// ---- 03_ControlPrimitives/Stamp/Stamp_StampWorkpiece.TcPOU
FUNCTION_BLOCK Stamp_StampWorkpiece EXTENDS ControlPrimitiveBase
VAR_INPUT
END_VAR
VAR_OUTPUT
END_VAR
VAR
	// (EProcessVariables.Stamp_WorkpieceState = 1) AND (EProcessVariables.Stamp_WPAtStamp = TRUE)
// 	m_compExpr273: ComparisonExpression(EProcessVariables.Stamp_WorkpieceState, EComparisonType.equals, EDataType.numeric, FALSE, 1, '', TRUE);
	m_precondition: ComparisonExpression(EProcessVariables.Stamp_WPAtStamp, EComparisonType.equals, EDataType.binary, TRUE, 0, '', TRUE);
// 	m_precondition: BoolExpression(m_compExpr273, EBoolOperation.and_op, m_compExpr275);
	
	// EProcessVariables.Stamp_WorkpieceState = 2
	m_postcondition: ComparisonExpression(EProcessVariables.Stamp_WorkpieceState, EComparisonType.equals, EDataType.numeric, FALSE, 2, '', TRUE);

	m_ptrStamp: POINTER TO Stamp;
	
	m_step: INT := 0;
	t_Stamp : TON;
END_VAR

SUPER^();

METHOD Abort : BOOL
VAR_INPUT
END_VAR
m_ptrStamp^.m_stampingCylinder.METH_Retract();
m_ptrStamp^.m_slidingCylinder.METH_Extend();
Abort := TRUE;
END_METHOD

(* Execution logic of this Control Primitive. *)
METHOD PROTECTED ExecuteInternal : BOOL
VAR_INPUT
	(*
	 * pressure_white: INT
	 * pressure_black: INT
	 * pressure_metal: INT
	 *)
	i_params: ParameterSet;
END_VAR
VAR
	m_pressureVal: SValue;
END_VAR
ExecuteInternal := FALSE;

CASE m_step OF
	0: // take in wp
	m_ptrStamp^.m_slidingCylinder.METH_Retract();
	IF m_ptrStamp^.m_slidingCylinder.Retracted THEN
		m_step := 1;
	END_IF
	
	1: // stamp wp
	m_ptrStamp^.StampPressure := GetPressure(i_params);
	m_ptrStamp^.m_stampingCylinder.METH_Extend();
	t_Stamp(IN:=TRUE, PT:=T#1500MS);
	IF t_Stamp.Q THEN
		IF m_ptrStamp^.StampPressure >= m_pressureVal.Value.Numeric THEN
			m_step := 2;
			t_Stamp(IN:=FALSE);
		END_IF
	END_IF
	
	2: // retract stamp
	m_ptrStamp^.m_stampingCylinder.METH_Retract();
	IF m_ptrStamp^.m_stampingCylinder.Retracted THEN
		m_step := 3;
	END_IF
	
	3: // provide wp
	m_ptrStamp^.m_slidingCylinder.METH_Extend();
	IF m_ptrStamp^.m_slidingCylinder.Extended THEN
		m_step := 0;
		ExecuteInternal := TRUE;
	END_IF
END_CASE
END_METHOD

METHOD FB_init : BOOL
VAR_INPUT
	bInitRetains : BOOL; // if TRUE, the retain variables are initialized (warm start / cold start)
	bInCopyCode : BOOL;  // if TRUE, the instance afterwards gets moved into the copy code (online change)
	
	i_ptrStamp: POINTER TO Stamp;
END_VAR
m_ptrStamp := i_ptrStamp;

m_id := EPrimitives.Stamp_StampWorkpiece;
m_timeout := T#200S;
m_paramDefinition := 'pressure_white:INT;pressure_black:INT;pressure_metal:INT;';

Precondition := m_precondition;
Postcondition := m_postcondition;
END_METHOD

METHOD PRIVATE GetPressure : INT
VAR_INPUT
	(*
	 * pressure_white: INT
	 * pressure_black: INT
	 * pressure_metal: INT
	 *)
	i_params: ParameterSet;
END_VAR
VAR
	m_pressureVal: SValue;
END_VAR
CASE LREAL_TO_UINT(m_st^.GetNumeric(EProcessVariables.Stamp_ProductType)) OF
	EProductTypes.white:
		m_pressureVal := i_params.Retrieve('pressure_white');
		GetPressure := LREAL_TO_INT(m_pressureVal.Value.Numeric);
	EProductTypes.black:
		m_pressureVal := i_params.Retrieve('pressure_black');
		GetPressure := LREAL_TO_INT(m_pressureVal.Value.Numeric);
	EProductTypes.metal:
		m_pressureVal := i_params.Retrieve('pressure_metal');
		GetPressure := LREAL_TO_INT(m_pressureVal.Value.Numeric);
	ELSE
		GetPressure := 0;
END_CASE
END_METHOD

END_FUNCTION_BLOCK

// ---- 05_HardwareControl/EquipmentModule/Stamps/Stamp.TcPOU
FUNCTION_BLOCK Stamp EXTENDS BaseComponent
VAR_INPUT
END_VAR
VAR_OUTPUT
END_VAR
VAR
	m_stampingCylinder: MonostableCylinder;
	m_slidingCylinder: BistableCylinder;
	m_pressureValve: PropotionalValve;
	
	m_presenceSensor: PresenceSensor;
	m_pressureSensor: PressureSensor;
END_VAR

PROPERTY StampPressure : INT
GET
StampPressure:=m_pressureSensor.Value;
END_GET
SET
m_pressureValve.Pressure := StampPressure;
END_SET
END_PROPERTY

PROPERTY WPAtStart : BOOL
GET
WPAtStart := m_presenceSensor.Value;
END_GET
END_PROPERTY

END_FUNCTION_BLOCK

// ---- 05_HardwareControl/ControlModule/Pushers/BistableCylinder.TcPOU
FUNCTION_BLOCK BistableCylinder EXTENDS BaseCylinder
VAR_INPUT	
END_VAR
VAR_OUTPUT
END_VAR
VAR	
	//Hardware
	DO_Retract AT %Q* : BOOL;
END_VAR

METHOD METH_Extend : BOOL
DO_Extend := TRUE;
DO_Retract := FALSE;
END_METHOD

METHOD METH_Retract : BOOL
DO_Extend := FALSE;
DO_Retract := TRUE;
END_METHOD

END_FUNCTION_BLOCK

// ---- 05_HardwareControl/ControlModule/Valves/PropotionalValve.TcPOU
FUNCTION_BLOCK PropotionalValve
VAR_INPUT
END_VAR
VAR_OUTPUT
END_VAR
VAR
	//Hardware
	AO_SetPressure AT %Q* : INT;
END_VAR

PROPERTY Pressure : INT
SET
AO_SetPressure := Pressure;
END_SET
END_PROPERTY

END_FUNCTION_BLOCK

// ---- 05_HardwareControl/ControlModule/Sensors/PressureSensor.TcPOU
FUNCTION_BLOCK PressureSensor IMPLEMENTS ITF_AnalogSensor
VAR_INPUT
END_VAR
VAR_OUTPUT
END_VAR
VAR
	//Hardware
	AI_CurrentPressure AT %I* : INT;
END_VAR

PROPERTY Value : INT
GET
Value := AI_CurrentPressure;
END_GET
END_PROPERTY

END_FUNCTION_BLOCK

// ---- 04_HardwareObservation/ObserveCrane.TcPOU
FUNCTION_BLOCK ObserveCrane EXTENDS HardwareObservationBase
VAR_INPUT
END_VAR
VAR_OUTPUT
END_VAR
VAR
	m_ptrCrane: POINTER TO Crane;
	m_ptrCraneWP: POINTER TO xPPUProduct;
	
	m_rtAtStack: R_TRIG;
	m_rtAtLSC: R_TRIG;
	m_rtAtStamp: R_TRIG;
	
	m_resetCranePos: BOOL;
	
	// needed for a regression for the analog AngleDeg
	poti0: REAL;
	poti90: REAL;
	poti180: REAL;
END_VAR

METHOD FB_init : BOOL
VAR_INPUT
	bInitRetains : BOOL; // if TRUE, the retain variables are initialized (warm start / cold start)
	bInCopyCode : BOOL;  // if TRUE, the instance afterwards gets moved into the copy code (online change)

	i_ptrCrane: POINTER TO Crane;
	i_ptrWP: POINTER TO xPPUProduct;
END_VAR
m_ptrCrane := i_ptrCrane;
m_ptrCraneWP := i_ptrWP;
END_METHOD

METHOD  ResetDefinition : BOOL
VAR_INPUT
END_VAR
m_resetCranePos := TRUE;
END_METHOD

(* Update an instance of ProcessState with the part of the process that can be observed by this Hardware Interface. *)
METHOD UpdateProcessObservation : BOOL
VAR_IN_OUT
	io_processState: ProcessState;
END_VAR
VAR
	potiVal: REAL;
	x_bar: REAL;
	y_bar: REAL;
	a: REAL := -88.16748;		// initial value (calibrated 30 April 2025)
	b: REAL := 0.0129453959;	// initial value (calibrated 30 April 2025)
END_VAR
io_processState.UpdateState_Binary(EProcessVariables.Crane_AtStack, m_ptrCrane^.AtStack, i_force := TRUE);
io_processState.UpdateState_Binary(EProcessVariables.Crane_AtStamp, m_ptrCrane^.AtStamp, i_force := TRUE);
io_processState.UpdateState_Binary(EProcessVariables.Crane_AtLSC, m_ptrCrane^.AtConveyor, i_force := TRUE);
io_processState.UpdateState_Binary(EProcessVariables.Crane_HoldingWorkpiece, m_ptrCrane^.o_VacuumGripper.WPTaken, i_force := TRUE);
io_processState.UpdateState_Binary(EProcessVariables.Crane_CylinderExtended, m_ptrCrane^.o_MonostableCylinder.Extended, i_force := TRUE);
io_processState.UpdateState_Binary(EProcessVariables.Crane_CylinderRetracted, m_ptrCrane^.o_MonostableCylinder.Retracted, i_force := TRUE);

// Angle [in degrees] regression
potiVal := m_ptrCrane^.Motor.AI_Position;
IF m_ptrCrane^.AtStack THEN
	poti0 := potiVal;
ELSIF m_ptrCrane^.AtConveyor THEN
	poti90 := potiVal;
ELSIF m_ptrCrane^.AtStamp THEN
	poti180 := potiVal;
END_IF

IF poti0 <> 0 AND poti90 <> 0 AND poti180 <> 0 THEN
	x_bar := (poti0 + poti90 + poti180) / 3;
	y_bar := (90+180)/3;
	b := ((poti0 - x_bar)*-y_bar + (poti90 - x_bar)*(90 - y_bar) + (poti180 - x_bar)*(180 - y_bar))/
		(EXPT(poti0 - x_bar, 2) + EXPT(poti90 - x_bar, 2) + EXPT(poti180 - x_bar, 2));
	a := y_bar - b*x_bar;
ELSIF poti0 <> 0 AND poti90 <> 0 THEN
	x_bar := (poti0 + poti90) / 2;
	y_bar := 90/2;
	b := ((poti0 - x_bar)*-y_bar + (poti90 - x_bar)*(90 - y_bar))/
		(EXPT(poti0 - x_bar, 2) + EXPT(poti90 - x_bar, 2));
	a := y_bar - b*x_bar;
ELSIF poti90 <> 0 AND poti180 <> 0 THEN
	x_bar := (poti90 + poti180) / 2;
	y_bar := (90+180)/2;
	b := ((poti90 - x_bar)*(90 - y_bar) + (poti180 - x_bar)*(180 - y_bar))/
		(EXPT(poti90 - x_bar, 2) + EXPT(poti180 - x_bar, 2));
	a := y_bar - b*x_bar;
END_IF

io_processState.UpdateState_Numeric(EProcessVariables.Crane_Angle, a + b*potiVal, i_force := TRUE);

m_rtAtStack(CLK := m_ptrCrane^.AtStack);
m_rtAtStamp(CLK := m_ptrCrane^.AtStamp);
m_rtAtLSC(CLK := m_ptrCrane^.AtConveyor);

IF m_rtAtStack.Q OR m_rtAtStamp.Q OR m_rtAtLSC.Q THEN
	io_processState.UpdateState_Defined(EProcessVariables.Crane_AtStack, TRUE);
	io_processState.UpdateState_Defined(EProcessVariables.Crane_AtStamp, TRUE);
	io_processState.UpdateState_Defined(EProcessVariables.Crane_AtLSC, TRUE);
END_IF
IF m_resetCranePos THEN
	io_processState.UpdateState_Defined(EProcessVariables.Crane_AtStack, FALSE);
	io_processState.UpdateState_Defined(EProcessVariables.Crane_AtStamp, FALSE);
	io_processState.UpdateState_Defined(EProcessVariables.Crane_AtLSC, FALSE);
	m_resetCranePos := FALSE;
END_IF

io_processState.UpdateState_Defined(EProcessVariables.Crane_HoldingWorkpiece, TRUE);
io_processState.UpdateState_Defined(EProcessVariables.Crane_CylinderExtended, TRUE);
io_processState.UpdateState_Defined(EProcessVariables.Crane_CylinderRetracted, TRUE);
io_processState.UpdateState_Defined(EProcessVariables.Crane_Angle, TRUE);
END_METHOD

END_FUNCTION_BLOCK

// ---- 04_HardwareObservation/xPPUProduct.TcPOU
FUNCTION_BLOCK xPPUProduct EXTENDS ProductBase
VAR CONSTANT
	LIGHT_IDX: USINT := 1;
	METAL_IDX: USINT := 2;
	PRESENT_IDX: USINT := 3;
	STAMPED_IDX: USINT := 4;

	LIGHT_MASK: BYTE := 2#0000_0001;
	METAL_MASK: BYTE := 2#0000_0010;
	PRESENT_MASK: BYTE := 2#0000_0100;
	STAMPED_MASK: BYTE := 2#0000_1000;
END_VAR
VAR
	m_productStampedIdx: UINT;
END_VAR

//FB_Init is always available implicitly and it is used primarily for initialization.
//The return value is not evaluated. For a specific influence, you can also declare the
//methods explicitly and provide additional code there with the standard initialization
//code. You can evaluate the return value.
METHOD FB_Init: BOOL
VAR_INPUT
    bInitRetains: BOOL; // TRUE: the retain variables are initialized (reset warm / reset cold)
    bInCopyCode: BOOL;  // TRUE: the instance will be copied to the copy code afterward (online change)
	
	i_productTypeVarId: UINT;
	i_productStampedVarId: UINT;
END_VAR
// set the variable indices (on remote, the RA does this)
raIn_processStateIdx := i_productTypeVarId;

m_productStampedIdx := i_productStampedVarId;

// set the variables' data types
m_vals[RES_IDX].DataType := EDataType.numeric;
m_vals[LIGHT_IDX].DataType := EDataType.binary;
m_vals[METAL_IDX].DataType := EDataType.binary;
m_vals[PRESENT_IDX].DataType := EDataType.binary;
END_METHOD

PROPERTY IsLight : BOOL
GET
IsLight := m_vals[LIGHT_IDX].Defined AND m_vals[LIGHT_IDX].Value.Binary;
END_GET
SET
m_vals[LIGHT_IDX].DataType := EDataType.binary;
m_vals[LIGHT_IDX].Defined := TRUE;
m_vals[LIGHT_IDX].Value.Binary := IsLight;

UpdateMaterial();
END_SET
END_PROPERTY

PROPERTY IsMetal : BOOL
GET
IsMetal := m_vals[METAL_IDX].Defined AND m_vals[METAL_IDX].Value.Binary;
END_GET
SET
m_vals[METAL_IDX].DataType := EDataType.binary;
m_vals[METAL_IDX].Defined := TRUE;
m_vals[METAL_IDX].Value.Binary := IsMetal;

UpdateMaterial();
END_SET
END_PROPERTY

PROPERTY IsPresent : BOOL
GET
IsPresent := m_vals[PRESENT_IDX].Defined AND m_vals[PRESENT_IDX].Value.Binary;
END_GET
SET
m_vals[PRESENT_IDX].DataType := EDataType.binary;
m_vals[PRESENT_IDX].Defined := TRUE;
m_vals[PRESENT_IDX].Value.Binary := IsPresent;

UpdateMaterial();
END_SET
END_PROPERTY

PROPERTY IsStamped : BOOL
GET
IsStamped := m_vals[STAMPED_IDX].Defined AND m_vals[STAMPED_IDX].Value.Binary;
END_GET
SET
m_vals[STAMPED_IDX].DataType := EDataType.binary;
m_vals[STAMPED_IDX].Defined := TRUE;
m_vals[STAMPED_IDX].Value.Binary := IsStamped;

UpdateMaterial();
END_SET
END_PROPERTY

(* Based on the aggregated product type value, set the separete input values for a consistent shift register. *)
METHOD ReverseSetInputs : BOOL
VAR
	res: BYTE;
END_VAR
res := LREAL_TO_BYTE(m_vals[RES_IDX].Value.Numeric);

m_vals[LIGHT_IDX].Value.Binary := (res AND LIGHT_MASK) <> 0;
m_vals[METAL_IDX].Value.Binary := (res AND METAL_MASK) <> 0;
m_vals[PRESENT_IDX].Value.Binary := (res AND PRESENT_MASK) <> 0;
m_vals[STAMPED_IDX].Value.Binary := (res AND STAMPED_MASK) <> 0;

m_vals[LIGHT_IDX].Defined := TRUE;
m_vals[METAL_IDX].Defined := TRUE;
m_vals[PRESENT_IDX].Defined := TRUE;
m_vals[STAMPED_IDX].Defined := TRUE;
END_METHOD

METHOD PRIVATE UpdateMaterial : BOOL
VAR
	res: BYTE;
END_VAR
// use separate bits to encode the product info
res := 2#0000_0000;

IF IsLight THEN
	res := res OR LIGHT_MASK;
END_IF
IF IsMetal THEN
	res := res OR METAL_MASK;
END_IF
IF IsPresent THEN
	res := res OR PRESENT_MASK;
END_IF
IF IsStamped THEN
	res := res OR STAMPED_MASK;
END_IF

m_vals[RES_IDX].DataType := EDataType.numeric;
m_vals[RES_IDX].Defined := TRUE;
m_vals[RES_IDX].Value.Numeric := BYTE_TO_LREAL(res);
END_METHOD

METHOD PROTECTED UpdateProcessObsInternal : BOOL
VAR_IN_OUT
	io_processState: ProcessState;
END_VAR
VAR
	prodType: EProductTypes;
END_VAR
IF NOT IsLight AND NOT IsMetal AND NOT IsPresent THEN
	prodType := EProductTypes.none;
ELSIF IsLight AND NOT IsMetal AND IsPresent THEN
	prodType := EProductTypes.white;
ELSIF NOT IsLight AND NOT IsMetal AND IsPresent THEN
	prodType := EProductTypes.black;
ELSIF IsMetal AND IsPresent THEN
	prodType := EProductTypes.metal;
END_IF

io_processState.UpdateState_Numeric(raIn_processStateIdx, UINT_TO_LREAL(prodType), i_force := TRUE);
io_processState.UpdateState_Binary(m_productStampedIdx, IsStamped, i_force := TRUE);

io_processState.UpdateState_Defined(raIn_processStateIdx, TRUE);
io_processState.UpdateState_Defined(m_productStampedIdx, TRUE);
END_METHOD

END_FUNCTION_BLOCK

// ---- 04_HardwareObservation/ObserveLSC.TcPOU
FUNCTION_BLOCK ObserveLSC EXTENDS HardwareObservationBase
VAR_INPUT
END_VAR
VAR_OUTPUT
END_VAR
VAR
	m_ptrLSC: POINTER TO LargeSortingConveyor;
	m_ptrLSCWP: POINTER TO xPPUProduct;
	
	m_rtAtStart: R_TRIG;
	m_rtLightAtStart: R_TRIG;
	m_rtLightAtMid: R_TRIG;
	m_rtLightAtEnd: R_TRIG;
	m_rtMetalAtStart: R_TRIG;
	m_rtMetalAtMid: R_TRIG;
	m_rtWpAtRampStart: R_TRIG;
	m_rtWpAtRampMiddle: R_TRIG;
	m_rtWpAtRampEnd: R_TRIG;
	
	m_LSCemptytimeout: TON;
	m_resetProductDefined: BOOL;
	
	m_didInit: BOOL := FALSE;
END_VAR

METHOD FB_init : BOOL
VAR_INPUT
	bInitRetains : BOOL; // if TRUE, the retain variables are initialized (warm start / cold start)
	bInCopyCode : BOOL;  // if TRUE, the instance afterwards gets moved into the copy code (online change)

	i_ptrLSC: POINTER TO LargeSortingConveyor;
	i_ptrWP: POINTER TO xPPUProduct;
END_VAR
m_ptrLSC := i_ptrLSC;
m_ptrLSCWP := i_ptrWP;
END_METHOD

METHOD  ResetDefinition : BOOL
VAR_INPUT
END_VAR
m_resetProductDefined := TRUE;
END_METHOD

(* Update an instance of ProcessState with the part of the process that can be observed by this Hardware Interface. *)
METHOD UpdateProcessObservation : BOOL
VAR_IN_OUT
	io_processState: ProcessState;
END_VAR
m_rtAtStart(CLK := m_ptrLSC^.WPAtStart);
m_rtLightAtStart(CLK := m_ptrLSC^.LightWPAtStart);
m_rtLightAtMid(CLK := m_ptrLSC^.LightWPAtMid);
m_rtLightAtEnd(CLK := m_ptrLSC^.LightWPAtEnd);
m_rtMetalAtStart(CLK := m_ptrLSC^.MetalWPAtStart);
m_rtMetalAtMid(CLK := m_ptrLSC^.MetalWPAtMid);
m_rtWpAtRampStart(CLK := m_ptrLSC^.WPAtRampStart);
m_rtWpAtRampMiddle(CLK := m_ptrLSC^.WPAtRampMiddle);
m_rtWpAtRampEnd(CLK := m_ptrLSC^.WPAtRampEnd);

io_processState.UpdateState_Binary(EProcessVariables.LSC_WorkpieceAtEntry, m_ptrLSC^.WPAtStart, TRUE);
io_processState.UpdateState_Binary(EProcessVariables.LSC_WPAtRampStart, m_ptrLSC^.WPAtRampStart, TRUE);
io_processState.UpdateState_Binary(EProcessVariables.LSC_WPAtRampMiddle, m_ptrLSC^.WPAtRampMiddle, TRUE);
io_processState.UpdateState_Binary(EProcessVariables.LSC_WPAtRampEnd, m_ptrLSC^.WPAtRampEnd, TRUE);
io_processState.UpdateState_Binary(EProcessVariables.LSC_SwitchExtended, m_ptrLSC^.m_Switch.Extended, TRUE);
io_processState.UpdateState_Binary(EProcessVariables.LSC_SwitchRetracted, m_ptrLSC^.m_Switch.Retracted, TRUE);
io_processState.UpdateState_Binary(EProcessVariables.LSC_WPAtInductiveSensorEnd, m_ptrLSC^.MetalWPAtMid, TRUE);

IF NOT m_didInit THEN
	io_processState.UpdateState_Numeric(EProcessVariables.LSC_RampStartWPCount, 0, TRUE);
	io_processState.UpdateState_Numeric(EProcessVariables.LSC_RampMiddleWPCount, 0, TRUE);
	io_processState.UpdateState_Numeric(EProcessVariables.LSC_RampEndWPCount, 0, TRUE);
	m_didInit := TRUE;
END_IF

IF m_rtWpAtRampStart.Q THEN
	io_processState.UpdateState_NumericIncrement(EProcessVariables.LSC_RampStartWPCount, TRUE);
END_IF
IF m_rtWpAtRampMiddle.Q THEN
	io_processState.UpdateState_NumericIncrement(EProcessVariables.LSC_RampMiddleWPCount, TRUE);
END_IF
IF m_rtWpAtRampEnd.Q THEN
	io_processState.UpdateState_NumericIncrement(EProcessVariables.LSC_RampEndWPCount, TRUE);
END_IF

io_processState.UpdateState_Defined(EProcessVariables.LSC_WorkpieceAtEntry, TRUE);
io_processState.UpdateState_Defined(EProcessVariables.LSC_WPAtRampStart, TRUE);
io_processState.UpdateState_Defined(EProcessVariables.LSC_WPAtRampMiddle, TRUE);
io_processState.UpdateState_Defined(EProcessVariables.LSC_WPAtRampEnd, TRUE);
io_processState.UpdateState_Defined(EProcessVariables.LSC_SwitchExtended, TRUE);
io_processState.UpdateState_Defined(EProcessVariables.LSC_SwitchRetracted, TRUE);
io_processState.UpdateState_Defined(EProcessVariables.LSC_WPAtInductiveSensorEnd, TRUE);
// TODO - the following are technically not defined but how can we avoid that?
io_processState.UpdateState_Defined(EProcessVariables.LSC_RampStartWPCount, TRUE);
io_processState.UpdateState_Defined(EProcessVariables.LSC_RampMiddleWPCount, TRUE);
io_processState.UpdateState_Defined(EProcessVariables.LSC_RampEndWPCount, TRUE);

// update WP info (if there are sensors available), then update the process variables list
IF m_rtAtStart.Q THEN
	m_ptrLSCWP^.IsPresent := TRUE;
END_IF
IF m_rtLightAtStart.Q OR m_rtLightAtMid.Q OR m_rtLightAtEnd.Q THEN
	m_ptrLSCWP^.IsLight := TRUE;
END_IF
IF m_rtMetalAtStart.Q OR m_rtMetalAtMid.Q THEN
	m_ptrLSCWP^.IsMetal := TRUE;
END_IF

// reset IsPresent if any of the ramps are triggered
IF m_ptrLSC^.WPAtRampStart OR m_ptrLSC^.WPAtRampMiddle OR m_ptrLSC^.WPAtRampEnd THEN
	m_ptrLSCWP^.IsPresent := FALSE;
END_IF

//if the conveyor moves forward for a certain time, it has to empty, therefore LSCProductType is defined
IF m_ptrLSC^.Motor.TurningClockwise THEN
	m_LSCemptytimeout(IN:= TRUE, PT:=T#3500MS);
ELSE
	m_LSCemptytimeout(IN:= FALSE);
END_IF

IF m_LSCemptytimeout.Q THEN
	io_processState.UpdateState_Defined(EProcessVariables.LSC_ProductType, TRUE);
	m_LSCemptytimeout(IN:= FALSE);
END_IF

IF m_resetProductDefined THEN
	m_resetProductDefined := TRUE;
END_IF
END_METHOD

END_FUNCTION_BLOCK

// ---- 04_HardwareObservation/ObservePAC.TcPOU
FUNCTION_BLOCK ObservePAC EXTENDS HardwareObservationBase
VAR_INPUT
END_VAR
VAR_OUTPUT
END_VAR
VAR
	m_ptrPAC: POINTER TO PicAlphaConveyor;
	m_ptrPACWP1: POINTER TO xPPUProduct;
	m_ptrPACWP2: POINTER TO xPPUProduct;
	m_ptrPACWP3: POINTER TO xPPUProduct;
END_VAR

METHOD FB_init : BOOL
VAR_INPUT
	bInitRetains : BOOL; // if TRUE, the retain variables are initialized (warm start / cold start)
	bInCopyCode : BOOL;  // if TRUE, the instance afterwards gets moved into the copy code (online change)
	
	i_ptrPAC: POINTER TO PicAlphaConveyor;
	i_ptrWP1: POINTER TO xPPUProduct;
	i_ptrWP2: POINTER TO xPPUProduct;
	i_ptrWP3: POINTER TO xPPUProduct;

	
END_VAR
m_ptrPAC := i_ptrPAC;
m_ptrPACWP1 := i_ptrWP1;
m_ptrPACWP2 := i_ptrWP2;
m_ptrPACWP3 := i_ptrWP3;
END_METHOD

METHOD  ResetDefinition : BOOL
VAR_INPUT
END_VAR
;
END_METHOD

(* Update an instance of ProcessState with the part of the process that can be observed by this Hardware Interface. *)
METHOD UpdateProcessObservation : BOOL
VAR_IN_OUT
	io_processState: ProcessState;
END_VAR
io_processState.UpdateState_Binary(EProcessVariables.PAC_WPAtStart, m_ptrPAC^.WPAtStart, TRUE);
io_processState.UpdateState_Binary(EProcessVariables.PAC_WPAtEnd, m_ptrPAC^.WPAtEnd, TRUE);
io_processState.UpdateState_Binary(EProcessVariables.PAC_SwitchExtended, m_ptrPAC^.m_Switch.Extended, TRUE);
io_processState.UpdateState_Binary(EProcessVariables.PAC_SwitchRetracted, m_ptrPAC^.m_Switch.Retracted, TRUE);
io_processState.UpdateState_Numeric(EProcessVariables.PAC_WPNumber, INT_TO_LREAL(m_ptrPAC^.m_WPNumberAtPAC), TRUE);

io_processState.UpdateState_Defined(EProcessVariables.PAC_WPAtStart, TRUE);
io_processState.UpdateState_Defined(EProcessVariables.PAC_WPAtEnd, TRUE);
io_processState.UpdateState_Defined(EProcessVariables.PAC_SwitchExtended, TRUE);
io_processState.UpdateState_Defined(EProcessVariables.PAC_SwitchRetracted, TRUE);
io_processState.UpdateState_Defined(EProcessVariables.PAC_WPNumber, TRUE);
END_METHOD

END_FUNCTION_BLOCK

// ---- 04_HardwareObservation/ObservePicAlpha.TcPOU
FUNCTION_BLOCK ObservePicAlpha EXTENDS HardwareObservationBase
VAR_INPUT
END_VAR
VAR_OUTPUT
END_VAR
VAR
	m_ptrPicAlpha: POINTER TO PicAlpha;
	m_ptrPicAlphaWP: POINTER TO xPPUProduct;

	m_PicAlphaPosDefinedState: BOOL := FALSE;
END_VAR

METHOD FB_init : BOOL
VAR_INPUT
	bInitRetains : BOOL; // if TRUE, the retain variables are initialized (warm start / cold start)
	bInCopyCode : BOOL;  // if TRUE, the instance afterwards gets moved into the copy code (online change)
	
	i_ptrPicAlpha: POINTER TO PicAlpha;
	i_ptrWP: POINTER TO xPPUProduct;
END_VAR
m_ptrPicAlpha := i_ptrPicAlpha;
m_ptrPicAlphaWP := i_ptrWP;
END_METHOD

METHOD  ResetDefinition : BOOL
VAR_INPUT
END_VAR
m_PicAlphaPosDefinedState := FALSE;
END_METHOD

(* Update an instance of ProcessState with the part of the process that can be observed by this Hardware Interface. *)
METHOD UpdateProcessObservation : BOOL
VAR_IN_OUT
	io_processState: ProcessState;
END_VAR
VAR
	m_sensorCount : UINT;
END_VAR
io_processState.UpdateState_Binary(EProcessVariables.PicAlpha_AtPos1, m_ptrPicAlpha^.PresenceSensorPosition1Value, i_force := TRUE);
io_processState.UpdateState_Binary(EProcessVariables.PicAlpha_AtPos2, m_ptrPicAlpha^.PresenceSensorPosition2Value, i_force := TRUE);
io_processState.UpdateState_Binary(EProcessVariables.PicAlpha_AtPos3, m_ptrPicAlpha^.PresenceSensorPosition3Value, i_force := TRUE);
io_processState.UpdateState_Binary(EProcessVariables.PicAlpha_AtPos4, m_ptrPicAlpha^.PresenceSensorPosition4Value, i_force := TRUE);
io_processState.UpdateState_Binary(EProcessVariables.PicAlpha_HoldingWorkpiece, m_ptrPicAlpha^.o_VacuumGripper.WPTaken, i_force := TRUE);
io_processState.UpdateState_Binary(EProcessVariables.PicAlpha_CylinderExtended, m_ptrPicAlpha^.o_MonostableCylinder.Extended, i_force := TRUE);
io_processState.UpdateState_Binary(EProcessVariables.PicAlpha_CylinderRetracted, m_ptrPicAlpha^.o_MonostableCylinder.Retracted, i_force := TRUE);
io_processState.UpdateState_Numeric(EProcessVariables.PicAlpha_Distance, INT_TO_LREAL(m_ptrPicAlpha^.o_Distance), i_force := TRUE);

io_processState.UpdateState_Defined(EProcessVariables.PicAlpha_HoldingWorkpiece, TRUE);
io_processState.UpdateState_Defined(EProcessVariables.PicAlpha_CylinderExtended, TRUE);
io_processState.UpdateState_Defined(EProcessVariables.PicAlpha_CylinderRetracted, TRUE);
io_processState.UpdateState_Defined(EProcessVariables.PicAlpha_Distance, TRUE);

// update WP info (if there are sensors available), then update the process variables list

IF m_ptrPicAlpha^.PresenceSensorPosition3Value AND NOT (m_ptrPicAlpha^.PresenceSensorPosition1Value OR m_ptrPicAlpha^.PresenceSensorPosition2Value OR m_ptrPicAlpha^.PresenceSensorPosition4Value) THEN
	m_PicAlphaPosDefinedState :=  TRUE;
END_IF
IF m_PicAlphaPosDefinedState THEN
	m_sensorCount := 0;	
END_IF
IF m_ptrPicAlpha^.PresenceSensorPosition1Value OR m_ptrPicAlpha^.PresenceSensorPosition2Value THEN
 	m_sensorCount := m_sensorCount + 1;
END_IF
IF m_ptrPicAlpha^.PresenceSensorPosition3Value THEN
 	m_sensorCount := m_sensorCount + 1;
END_IF
IF m_ptrPicAlpha^.PresenceSensorPosition4Value THEN
 	m_sensorCount := m_sensorCount + 1;
END_IF

IF m_sensorCount > 1 THEN // if more than one sensor is pressed at the same time, the position is undefined
	m_PicAlphaPosDefinedState := FALSE;	
END_IF

io_processState.UpdateState_Defined(EProcessVariables.PicAlpha_AtPos1, m_PicAlphaPosDefinedState);
io_processState.UpdateState_Defined(EProcessVariables.PicAlpha_AtPos2, m_PicAlphaPosDefinedState);
io_processState.UpdateState_Defined(EProcessVariables.PicAlpha_AtPos3, m_PicAlphaPosDefinedState);
io_processState.UpdateState_Defined(EProcessVariables.PicAlpha_AtPos4, m_PicAlphaPosDefinedState);
END_METHOD

END_FUNCTION_BLOCK

// ---- 04_HardwareObservation/ObserveRFC.TcPOU
FUNCTION_BLOCK ObserveRFC
VAR_INPUT
END_VAR
VAR_OUTPUT
END_VAR
VAR
	m_ptrRFC: POINTER TO RefeedingConveyor;
	m_ptrRFCWP1: POINTER TO xPPUProduct;
	m_ptrRFCWP2: POINTER TO xPPUProduct;
END_VAR

METHOD FB_init : BOOL
VAR_INPUT
	bInitRetains : BOOL; // if TRUE, the retain variables are initialized (warm start / cold start)
	bInCopyCode : BOOL;  // if TRUE, the instance afterwards gets moved into the copy code (online change)
	
	i_ptrRFC: POINTER TO RefeedingConveyor;
	i_ptrWP1: POINTER TO xPPUProduct;
	i_ptrWP2: POINTER TO xPPUProduct;
END_VAR
m_ptrRFC := i_ptrRFC;
m_ptrRFCWP1 := i_ptrWP1;
m_ptrRFCWP2 := i_ptrWP2;
END_METHOD

METHOD ResetDefinition : BOOL
VAR_INPUT
END_VAR
;
END_METHOD

(* Update an instance of ProcessState with the part of the process that can be observed by this Hardware Interface. *)
METHOD UpdateProcessObservation : BOOL
VAR_IN_OUT
	io_processState: ProcessState;
END_VAR
io_processState.UpdateState_Binary(EProcessVariables.RFC_WPAtStart, m_ptrRFC^.WPAtStart, TRUE);
io_processState.UpdateState_Binary(EProcessVariables.RFC_WPAtEnd, m_ptrRFC^.WPAtEnd, TRUE);
io_processState.UpdateState_Binary(EProcessVariables.RFC_SwitchExtended, m_ptrRFC^.m_Switch.Extended, TRUE);
io_processState.UpdateState_Binary(EProcessVariables.RFC_SwitchRetracted, m_ptrRFC^.m_Switch.Retracted, TRUE);

io_processState.UpdateState_Defined(EProcessVariables.RFC_WPAtStart, TRUE);
io_processState.UpdateState_Defined(EProcessVariables.RFC_WPAtEnd, TRUE);
io_processState.UpdateState_Defined(EProcessVariables.RFC_SwitchExtended, TRUE);
io_processState.UpdateState_Defined(EProcessVariables.RFC_SwitchRetracted, TRUE);
END_METHOD

END_FUNCTION_BLOCK

// ---- 04_HardwareObservation/ObserveSSC.TcPOU
FUNCTION_BLOCK ObserveSSC EXTENDS HardwareObservationBase
VAR_INPUT
END_VAR
VAR_OUTPUT
END_VAR
VAR
	m_ptrSSC: POINTER TO SmallSortingConveyor;
	m_ptrSSCWP1: POINTER TO xPPUProduct;
	m_ptrSSCWP2: POINTER TO xPPUProduct;
	
	m_rtWpAtRamp: R_TRIG;
END_VAR

METHOD FB_init : BOOL
VAR_INPUT
	bInitRetains : BOOL; // if TRUE, the retain variables are initialized (warm start / cold start)
	bInCopyCode : BOOL;  // if TRUE, the instance afterwards gets moved into the copy code (online change)
	
	i_ptrSSC: POINTER TO SmallSortingConveyor;
	i_ptrWP1: POINTER TO xPPUProduct;
	i_ptrWP2: POINTER TO xPPUProduct;
END_VAR
m_ptrSSC := i_ptrSSC;
m_ptrSSCWP1 := i_ptrWP1;
m_ptrSSCWP2 := i_ptrWP2;
END_METHOD

METHOD  ResetDefinition : BOOL
VAR_INPUT
END_VAR
;
END_METHOD

(* Update an instance of ProcessState with the part of the process that can be observed by this Hardware Interface. *)
METHOD UpdateProcessObservation : BOOL
VAR_IN_OUT
	io_processState: ProcessState;
END_VAR
m_rtWpAtRamp(CLK := m_ptrSSC^.WPAtRampEnd);

io_processState.UpdateState_Binary(EProcessVariables.SSC_WPAtStart, m_ptrSSC^.WPAtStart, TRUE);
io_processState.UpdateState_Binary(EProcessVariables.SSC_WPAtEnd, m_ptrSSC^.WPAtEnd, TRUE);
io_processState.UpdateState_Binary(EProcessVariables.SSC_WPLightAtMiddle, m_ptrSSC^.LightWPAtMid, TRUE);
io_processState.UpdateState_Binary(EProcessVariables.SSC_WPMetalAtMiddle, m_ptrSSC^.MetalWPAtMid, TRUE);
io_processState.UpdateState_Binary(EProcessVariables.SSC_WPAtRampEnd, m_ptrSSC^.WPAtRampEnd, TRUE);
io_processState.UpdateState_Binary(EProcessVariables.SSC_SwitchExtended, m_ptrSSC^.m_Switch.Extended, TRUE);
io_processState.UpdateState_Binary(EProcessVariables.SSC_SwitchRetracted, m_ptrSSC^.m_Switch.Retracted, TRUE);

IF m_rtWpAtRamp.Q THEN
	io_processState.UpdateState_NumericIncrement(EProcessVariables.SSC_RampWPCount, TRUE);
END_IF


io_processState.UpdateState_Defined(EProcessVariables.SSC_WPAtStart, TRUE);
io_processState.UpdateState_Defined(EProcessVariables.SSC_WPAtEnd, TRUE);
io_processState.UpdateState_Defined(EProcessVariables.SSC_WPLightAtMiddle, TRUE);
io_processState.UpdateState_Defined(EProcessVariables.SSC_WPMetalAtMiddle, TRUE);
io_processState.UpdateState_Defined(EProcessVariables.SSC_WPAtRampEnd, TRUE);
io_processState.UpdateState_Defined(EProcessVariables.SSC_SwitchExtended, TRUE);
io_processState.UpdateState_Defined(EProcessVariables.SSC_SwitchRetracted, TRUE);
// TODO - the following is technically not defined but how can we avoid that?
io_processState.UpdateState_Defined(EProcessVariables.SSC_RampWPCount, TRUE);
END_METHOD

END_FUNCTION_BLOCK

// ---- 04_HardwareObservation/ObserveStack.TcPOU
FUNCTION_BLOCK ObserveStack EXTENDS HardwareObservationBase
VAR_INPUT
END_VAR
VAR_OUTPUT
END_VAR
VAR
	m_ptrStack: POINTER TO Stack;
	m_ptrStackWP: POINTER TO xPPUProduct;
END_VAR

METHOD FB_init : BOOL
VAR_INPUT
	bInitRetains : BOOL; // if TRUE, the retain variables are initialized (warm start / cold start)
	bInCopyCode : BOOL;  // if TRUE, the instance afterwards gets moved into the copy code (online change)

	i_ptrStack: POINTER TO Stack;
	i_ptrWP: POINTER TO xPPUProduct;
END_VAR
m_ptrStack := i_ptrStack;
m_ptrStackWP := i_ptrWP;
END_METHOD

METHOD  ResetDefinition : BOOL
VAR_INPUT
END_VAR
;
END_METHOD

(* Update an instance of ProcessState with the part of the process that can be observed by this Hardware Interface. *)
METHOD UpdateProcessObservation : BOOL
VAR_IN_OUT
	io_processState: ProcessState;
END_VAR
io_processState.UpdateState_Binary(EProcessVariables.Stack_WorkpieceAvailable, m_ptrStack^.WPOnTray, i_force := TRUE);
io_processState.UpdateState_Binary(EProcessVariables.Stack_CylinderExtended, m_ptrStack^.o_slidingCylinder.Extended, i_force := TRUE);
io_processState.UpdateState_Binary(EProcessVariables.Stack_CylinderRetracted, m_ptrStack^.o_slidingCylinder.Retracted, i_force := TRUE);

io_processState.UpdateState_Defined(EProcessVariables.Stack_WorkpieceAvailable, TRUE);
io_processState.UpdateState_Defined(EProcessVariables.Stack_CylinderExtended, TRUE);
io_processState.UpdateState_Defined(EProcessVariables.Stack_CylinderRetracted, TRUE);

// update WP info (if there are sensors available), then update the process variables list
m_ptrStackWP^.IsPresent := m_ptrStack^.WPOnTray;
m_ptrStackWP^.IsLight := m_ptrStack^.LightWPOnTray;
m_ptrStackWP^.IsMetal := m_ptrStack^.MetalWPOnTray;
END_METHOD

END_FUNCTION_BLOCK

// ---- 04_HardwareObservation/ObserveStamp.TcPOU
FUNCTION_BLOCK ObserveStamp EXTENDS HardwareObservationBase
VAR_INPUT
END_VAR
VAR_OUTPUT
END_VAR
VAR
	m_ptrStamp: POINTER TO Stamp;
	m_ptrStampWP: POINTER TO xPPUProduct;
	m_detectionStep: INT := 0;
END_VAR

METHOD FB_init : BOOL
VAR_INPUT
	bInitRetains : BOOL; // if TRUE, the retain variables are initialized (warm start / cold start)
	bInCopyCode : BOOL;  // if TRUE, the instance afterwards gets moved into the copy code (online change)

	i_ptrStamp: POINTER TO Stamp;
	i_ptrWP: POINTER TO xPPUProduct;
END_VAR
m_ptrStamp := i_ptrStamp;
m_ptrStampWP := i_ptrWP;
END_METHOD

METHOD  ResetDefinition : BOOL
VAR_INPUT
END_VAR
;
END_METHOD

(* Update an instance of ProcessState with the part of the process that can be observed by this Hardware Interface. *)
METHOD UpdateProcessObservation : BOOL
VAR_IN_OUT
	io_processState: ProcessState;
END_VAR
io_processState.UpdateState_Binary(EProcessVariables.Stamp_StamperExtended, m_ptrStamp^.m_stampingCylinder.Extended, i_force := TRUE);
io_processState.UpdateState_Binary(EProcessVariables.Stamp_StamperRetracted, m_ptrStamp^.m_stampingCylinder.Retracted, i_force := TRUE);
io_processState.UpdateState_Binary(EProcessVariables.Stamp_SliderExtended, m_ptrStamp^.m_slidingCylinder.Extended, i_force := TRUE);
io_processState.UpdateState_Binary(EProcessVariables.Stamp_SliderRetracted, m_ptrStamp^.m_slidingCylinder.Retracted, i_force := TRUE);

io_processState.UpdateState_Binary(EProcessVariables.Stamp_WPAtStamp, m_ptrStamp^.WPAtStart, i_force := TRUE);
m_ptrStampWP^.IsPresent := m_ptrStamp^.WPAtStart;

CASE m_detectionStep OF
	0: // initial, empty state
	io_processState.UpdateState_Numeric(EProcessVariables.Stamp_WorkpieceState, EStampStates.none, i_force := TRUE);
	m_ptrStampWP^.IsStamped := FALSE;
	IF m_ptrStamp^.WPAtStart THEN
		m_detectionStep := 1;
	END_IF
	
	1: // WP received
	io_processState.UpdateState_Numeric(EProcessVariables.Stamp_WorkpieceState, EStampStates.unpressed, i_force := TRUE);
	IF NOT m_ptrStamp^.m_slidingCylinder.Extended THEN
		m_detectionStep := 2;
	ELSIF NOT m_ptrStamp^.WPAtStart THEN
		// WP removed without stamping
		m_detectionStep := 0;
	END_IF
	
	2: // busy
	io_processState.UpdateState_Numeric(EProcessVariables.Stamp_WorkpieceState, EStampStates.busy, i_force := TRUE);
	IF m_ptrStamp^.m_slidingCylinder.Extended THEN
		m_detectionStep := 3;
	END_IF
	
	3: // finished processing
	io_processState.UpdateState_Numeric(EProcessVariables.Stamp_WorkpieceState, EStampStates.pressed, i_force := TRUE);
	m_ptrStampWP^.IsStamped := TRUE;
	IF NOT m_ptrStamp^.WPAtStart THEN
		m_detectionStep := 0;
	END_IF
	
END_CASE

io_processState.UpdateState_Defined(EProcessVariables.Stamp_WPAtStamp, TRUE);
io_processState.UpdateState_Defined(EProcessVariables.Stamp_WorkpieceState, TRUE);
io_processState.UpdateState_Defined(EProcessVariables.Stamp_StamperExtended, TRUE);
io_processState.UpdateState_Defined(EProcessVariables.Stamp_StamperRetracted, TRUE);
io_processState.UpdateState_Defined(EProcessVariables.Stamp_SliderExtended, TRUE);
io_processState.UpdateState_Defined(EProcessVariables.Stamp_SliderRetracted, TRUE);
END_METHOD

END_FUNCTION_BLOCK

// ---- 99_ExtrafunctionalImpl/PanelManager.TcPOU
FUNCTION_BLOCK PanelManager EXTENDS HardwareObservationBase
VAR_INPUT
END_VAR
VAR_OUTPUT
END_VAR
VAR
	DI_StartBtn AT%I*: BOOL;
	DI_ModeSwitch AT%I*: BOOL;
	DI_EStopBtn AT%I*: BOOL;
	
	// only on safety panels
	DI_StopBtn AT%I*: BOOL;
	DI_ResetBtn AT%I*: BOOL;
	
	DO_GreenLight AT%Q*: BOOL;
	DO_WhiteLight AT%Q*: BOOL;	// on safety panels, this is the reset light
	
	// only on old panels
	DO_RedLight AT%Q*: BOOL;
	
	m_ptrSt: POINTER TO StateTracker;
	m_resetDefinitions: BOOL;
	
	m_startBtnIdx: UINT;
	m_stopBtnIdx: UINT;
	m_modeIdx: UINT;
	m_eStopBtnIdx: UINT;
	m_resetBtnIdx: UINT;
	
	// blink timers
	m_greenTmr: TON;
	m_redTmr: TON;
	m_whiteTmr: TON;
END_VAR

PROPERTY EStop : BOOL
GET
EStop := m_ptrSt^.GetBinary(EProcessVariables.Pnl_Stack_EStop)
	OR m_ptrSt^.GetBinary(EProcessVariables.Pnl_LSC_EStop)
	OR m_ptrSt^.GetBinary(EProcessVariables.Pnl_Stamp_EStop)
	OR m_ptrSt^.GetBinary(EProcessVariables.Pnl_LightBarrier_EStop)
	OR m_ptrSt^.GetBinary(EProcessVariables.Pnl_Door_EStop);
END_GET
END_PROPERTY

//FB_Init is always available implicitly and it is used primarily for initialization.
//The return value is not evaluated. For a specific influence, you can also declare the
//methods explicitly and provide additional code there with the standard initialization
//code. You can evaluate the return value.
METHOD FB_Init: BOOL
VAR_INPUT
    bInitRetains: BOOL; // TRUE: the retain variables are initialized (reset warm / reset cold)
    bInCopyCode: BOOL;  // TRUE: the instance will be copied to the copy code afterward (online change)
	
	i_ptrStateTracker: POINTER TO StateTracker;
	
	i_startBtnIdx: UINT;
	i_stopBtnIdx: UINT;
	i_modeIdx: UINT;
	i_eStopBtnIdx: UINT;
	i_resetBtnIdx: UINT;
END_VAR
m_ptrSt := i_ptrStateTracker;

m_startBtnIdx := i_startBtnIdx;
m_stopBtnIdx := i_stopBtnIdx;
m_modeIdx := i_modeIdx;
m_eStopBtnIdx := i_eStopBtnIdx;
m_resetBtnIdx := i_resetBtnIdx;
END_METHOD

PROPERTY Mode : EOperatingModes
GET
VAR
	m_isAuto: BOOL;
	m_isManu: BOOL;
END_VAR
m_isAuto :=
	(m_ptrSt^.GetNumeric(EProcessVariables.Pnl_Stack_Mode) = EOperatingModes.automatic OR NOT m_ptrSt^.GetDefined(EProcessVariables.Pnl_Stack_Mode))
	AND (m_ptrSt^.GetNumeric(EProcessVariables.Pnl_LSC_Mode) = EOperatingModes.automatic OR NOT m_ptrSt^.GetDefined(EProcessVariables.Pnl_LSC_Mode))
	AND (m_ptrSt^.GetNumeric(EProcessVariables.Pnl_Stamp_Mode) = EOperatingModes.automatic OR NOT m_ptrSt^.GetDefined(EProcessVariables.Pnl_Stamp_Mode))
	AND (m_ptrSt^.GetNumeric(EProcessVariables.Pnl_LightBarrier_Mode) = EOperatingModes.automatic OR NOT m_ptrSt^.GetDefined(EProcessVariables.Pnl_LightBarrier_Mode))
	AND (m_ptrSt^.GetNumeric(EProcessVariables.Pnl_Door_Mode) = EOperatingModes.automatic OR NOT m_ptrSt^.GetDefined(EProcessVariables.Pnl_Door_Mode));

m_isManu :=
	(m_ptrSt^.GetNumeric(EProcessVariables.Pnl_Stack_Mode) = EOperatingModes.manual OR NOT m_ptrSt^.GetDefined(EProcessVariables.Pnl_Stack_Mode))
	AND (m_ptrSt^.GetNumeric(EProcessVariables.Pnl_LSC_Mode) = EOperatingModes.manual OR NOT m_ptrSt^.GetDefined(EProcessVariables.Pnl_LSC_Mode))
	AND (m_ptrSt^.GetNumeric(EProcessVariables.Pnl_Stamp_Mode) = EOperatingModes.manual OR NOT m_ptrSt^.GetDefined(EProcessVariables.Pnl_Stamp_Mode))
	AND (m_ptrSt^.GetNumeric(EProcessVariables.Pnl_LightBarrier_Mode) = EOperatingModes.manual OR NOT m_ptrSt^.GetDefined(EProcessVariables.Pnl_LightBarrier_Mode))
	AND (m_ptrSt^.GetNumeric(EProcessVariables.Pnl_Door_Mode) = EOperatingModes.manual OR NOT m_ptrSt^.GetDefined(EProcessVariables.Pnl_Door_Mode));

IF m_isAuto THEN
	Mode := EOperatingModes.automatic;
ELSIF m_isManu THEN
	Mode := EOperatingModes.manual;
ELSE
	Mode := EOperatingModes.none;
END_IF
END_GET
END_PROPERTY

PROPERTY Reset : BOOL
GET
Reset := m_ptrSt^.GetBinary(EProcessVariables.Pnl_Door_Reset) OR m_ptrSt^.GetBinary(EProcessVariables.Pnl_LightBarrier_Reset);
END_GET
END_PROPERTY

METHOD ResetDefinition : BOOL
m_resetDefinitions := TRUE;
END_METHOD

METHOD SetGreen : BOOL
VAR_INPUT
	i_lightVal: BOOL;
	i_blinkTime: TIME := T#0S;	// blink state change time; 0 means constant on/off
END_VAR
IF i_blinkTime = T#0S THEN
	DO_GreenLight  := i_lightVal;
ELSE
	m_greenTmr(IN := TRUE, PT := i_blinkTime);
	IF m_greenTmr.Q THEN
		m_greenTmr(IN := FALSE);
		DO_GreenLight := NOT DO_GreenLight;
	END_IF
END_IF
END_METHOD

METHOD SetRed : BOOL
VAR_INPUT
	i_lightVal: BOOL;
	i_blinkTime: TIME := T#0S;	// blink state change time; 0 means constant on/off
END_VAR
IF i_blinkTime = T#0S THEN
	DO_RedLight  := i_lightVal;
ELSE
	m_redTmr(IN := TRUE, PT := i_blinkTime);
	IF m_redTmr.Q THEN
		m_redTmr(IN := FALSE);
		DO_RedLight := NOT DO_RedLight;
	END_IF
END_IF
END_METHOD

METHOD SetWhite : BOOL
VAR_INPUT
	i_lightVal: BOOL;
	i_blinkTime: TIME := T#0S;	// blink state change time; 0 means constant on/off
END_VAR
IF i_blinkTime = T#0S THEN
	DO_WhiteLight  := i_lightVal;
ELSE
	m_whiteTmr(IN := TRUE, PT := i_blinkTime);
	IF m_whiteTmr.Q THEN
		m_whiteTmr(IN := FALSE);
		DO_WhiteLight := NOT DO_WhiteLight;
	END_IF
END_IF
END_METHOD

PROPERTY Start : BOOL
GET
Start := 
	m_ptrSt^.GetBinary(EProcessVariables.Pnl_Stack_Start)
	OR m_ptrSt^.GetBinary(EProcessVariables.Pnl_LSC_Start)
	OR m_ptrSt^.GetBinary(EProcessVariables.Pnl_Stamp_Start)
	OR m_ptrSt^.GetBinary(EProcessVariables.Pnl_LightBarrier_Start)
	OR m_ptrSt^.GetBinary(EProcessVariables.Pnl_Door_Start);
END_GET
END_PROPERTY

PROPERTY Stop : BOOL
GET
Stop := m_ptrSt^.GetBinary(EProcessVariables.Pnl_LightBarrier_Stop)
	OR m_ptrSt^.GetBinary(EProcessVariables.Pnl_Door_Stop);
END_GET
END_PROPERTY

(* Update an instance of ProcessState with the part of the process that can be observed by this Hardware Interface. *)
METHOD UpdateProcessObservation : BOOL
VAR_IN_OUT
	io_processState: ProcessState;
END_VAR
IF m_startBtnIdx <> 0 THEN
	io_processState.UpdateState_Binary(m_startBtnIdx, DI_StartBtn, TRUE);
	io_processState.UpdateState_Defined(m_startBtnIdx, NOT m_resetDefinitions);
END_IF
IF m_stopBtnIdx <> 0 THEN
	// invert the EStop signal
	io_processState.UpdateState_Binary(m_stopBtnIdx, NOT DI_StopBtn, TRUE);
	io_processState.UpdateState_Defined(m_stopBtnIdx, NOT m_resetDefinitions);
END_IF
IF m_modeIdx <> 0 THEN
	IF DI_ModeSwitch THEN
		io_processState.UpdateState_Numeric(m_modeIdx, EOperatingModes.automatic, TRUE);
	ELSE
		io_processState.UpdateState_Numeric(m_modeIdx, EOperatingModes.manual, TRUE);
	END_IF
	io_processState.UpdateState_Defined(m_modeIdx, NOT m_resetDefinitions);
END_IF
IF m_eStopBtnIdx <> 0 THEN
	// invert the EStop signal
	io_processState.UpdateState_Binary(m_eStopBtnIdx, NOT DI_EStopBtn, TRUE);
	io_processState.UpdateState_Defined(m_eStopBtnIdx, NOT m_resetDefinitions);
END_IF
IF m_resetBtnIdx <> 0 THEN
	io_processState.UpdateState_Binary(m_resetBtnIdx, DI_ResetBtn, TRUE);
	io_processState.UpdateState_Defined(m_resetBtnIdx, NOT m_resetDefinitions);
END_IF

IF m_resetDefinitions THEN
	m_resetDefinitions := FALSE;
END_IF
END_METHOD

END_FUNCTION_BLOCK

// ---- 99_ExtrafunctionalImpl/ErrorManager.TcPOU
FUNCTION_BLOCK ErrorManager EXTENDS ErrorManagerBase
VAR CONSTANT
	ALARMS_ARR_MIN: UINT := 0;
	ALARMS_ARR_MAX: UINT := 9;
END_VAR
VAR
	{attribute 'OPC.UA.DA' := '1'}
	{attribute 'OPC.UA.DA.Access' := '1'}
	alarms: ARRAY [ALARMS_ARR_MIN..ALARMS_ARR_MAX] OF SAlarm;
END_VAR

METHOD AddMessage : BOOL
VAR_INPUT
	i_alarmId	: UINT;
	i_active	: BOOL;
	//i_acknowledged	: BOOL;
	//i_confirmed	: BOOL;
	i_severity	: ESeverity;
	//i_retain	: BOOL;
	i_instanceName: STRING;
	i_detailText: STRING := '';
END_VAR
VAR
	i: UINT;
END_VAR
// move all errors to next index
FOR i := ALARMS_ARR_MAX TO ALARMS_ARR_MIN + 1 BY -1  DO
	alarms[i] := alarms[i - 1];
END_FOR

// add new error at index 0
alarms[0].TimeTicks := F_GetSystemTime();
alarms[0].AlarmId := i_alarmId;
alarms[0].Active := i_active;
//alarms[0].Acknowledged := i_acknowledged;
//alarms[0].Confirmed := i_confirmed;
alarms[0].Severity := i_severity;
//alarms[0].RetainAlarm := i_retain;

IF LEN(i_detailText) > 0 THEN
	alarms[0].Message := CONCAT(CONCAT(HMI_Texts.AlarmTexts[i_alarmId], ': '), i_detailText);
ELSE
	alarms[0].Message := HMI_Texts.AlarmTexts[i_alarmId];
END_IF

alarms[0].InstanceName := i_instanceName;
END_METHOD

END_FUNCTION_BLOCK

// ---- 99_ExtrafunctionalImpl/FC_InitAlarmTexts.TcPOU
FUNCTION FC_InitAlarmTexts : BOOL
VAR_INPUT
END_VAR
VAR
END_VAR

HMI_Texts.AlarmTexts[EAlarms.none] := 'unspecified';
HMI_Texts.AlarmTexts[EAlarms.initialized] := 'the application is initialized';
HMI_Texts.AlarmTexts[EAlarms.did_execute] := 'the component executed';
HMI_Texts.AlarmTexts[EAlarms.stopped] := 'all operations stopped';
HMI_Texts.AlarmTexts[EAlarms.stopping] := 'finishing all Control Primitives';
HMI_Texts.AlarmTexts[EAlarms.aborting] := 'aborting all Control Primitives';

HMI_Texts.AlarmTexts[ESpecialAlarmIds.recovery_request] := 'a recovery was requested; stopping operations';
HMI_Texts.AlarmTexts[ESpecialAlarmIds.definition_request] := 'a definition was requested';
HMI_Texts.AlarmTexts[ESpecialAlarmIds.strategy_received] := 'starting new strategy';
HMI_Texts.AlarmTexts[ESpecialAlarmIds.interlock_violated] := 'interlock violated';

END_FUNCTION

// ---- 99_ExtrafunctionalImpl/MachineModes.TcPOU
FUNCTION_BLOCK MachineModes
VAR
	m_ptrServices: POINTER TO ServiceContainer;
	m_ptrPanelMgr: POINTER TO PanelManager;	

	m_stratState: EOperationResult;
	m_allFinished: BOOL;
	m_ton: TON;
END_VAR

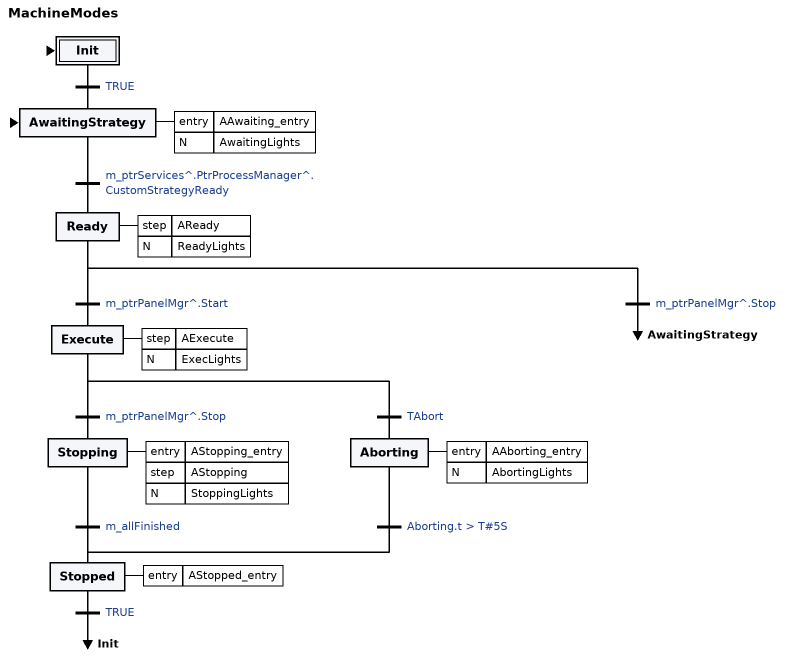
INITIAL_STEP Init:
END_STEP
TRANSITION FROM Init TO AwaitingStrategy
    := TRUE;
END_TRANSITION
STEP AwaitingStrategy:
    AAwaiting_entry(P1);  // entry action
    AwaitingLights(N);
END_STEP
TRANSITION FROM AwaitingStrategy TO Ready
    := m_ptrServices^.PtrProcessManager^.CustomStrategyReady;
END_TRANSITION
STEP Ready:
    AReady(N);  // step action
    ReadyLights(N);
END_STEP
TRANSITION FROM Ready TO Execute
    := m_ptrPanelMgr^.Start;
END_TRANSITION
TRANSITION FROM Ready TO AwaitingStrategy
    := m_ptrPanelMgr^.Stop;
END_TRANSITION
STEP Execute:
    AExecute(N);  // step action
    ExecLights(N);
END_STEP
TRANSITION FROM Execute TO Stopping
    := m_ptrPanelMgr^.Stop;
END_TRANSITION
STEP Stopping:
    AStopping_entry(P1);  // entry action
    AStopping(N);  // step action
    StoppingLights(N);
END_STEP
TRANSITION FROM Stopping TO Stopped
    := m_allFinished;
END_TRANSITION
TRANSITION FROM Execute TO Aborting
    := TAbort;
END_TRANSITION
STEP Aborting:
    AAborting_entry(P1);  // entry action
    AbortingLights(N);
END_STEP
TRANSITION FROM Aborting TO Stopped
    := Aborting.t > T#5S;
END_TRANSITION
STEP Stopped:
    AStopped_entry(P1);  // entry action
END_STEP
TRANSITION FROM Stopped TO Init
    := TRUE;
END_TRANSITION

ACTION AAborting_entry:
m_ptrServices^.PtrProcessManager^.RequestAbort();
m_ptrServices^.PtrErrorManager^.AddMessage(EAlarms.aborting, TRUE, ESeverity.info, 'Main');
END_ACTION

ACTION AAwaiting_entry:
m_ptrServices^.PtrErrorManager^.AddMessage(EAlarms.initialized, TRUE, ESeverity.info, 'Main');
END_ACTION

ACTION AbortingLights:
m_ptrPanelMgr^.SetGreen(FALSE);
m_ptrPanelMgr^.SetRed(TRUE, T#200MS);
m_ptrPanelMgr^.SetWhite(FALSE);
END_ACTION

ACTION AExecute:
m_stratState := m_ptrServices^.PtrProcessManager^.ExecuteCustomStrategy();
END_ACTION

ACTION AReady:
// TODO - blink light or something...
END_ACTION

ACTION AStopped_entry:
m_ptrServices^.PtrProcessManager^.ResetConfiguration();
m_ptrServices^.PtrStateTracker^.ResetConfiguration();
m_ptrServices^.PtrErrorManager^.AddMessage(EAlarms.stopped, TRUE, ESeverity.info, 'Main');
END_ACTION

ACTION AStopping:
m_allFinished := m_ptrServices^.PtrProcessManager^.FinishPrimitives(TRUE);
END_ACTION

ACTION AStopping_entry:
m_ptrServices^.PtrErrorManager^.AddMessage(EAlarms.stopping, TRUE, ESeverity.info, 'Main');
END_ACTION

ACTION AwaitingLights:
m_ptrPanelMgr^.SetGreen(FALSE);
m_ptrPanelMgr^.SetRed(FALSE);
m_ptrPanelMgr^.SetWhite(TRUE, T#500MS);
END_ACTION

ACTION ExecLights:
m_ptrPanelMgr^.SetGreen(TRUE);
m_ptrPanelMgr^.SetRed(FALSE);
m_ptrPanelMgr^.SetWhite(FALSE);
END_ACTION

//FB_Init is always available implicitly and it is used primarily for initialization.
//The return value is not evaluated. For a specific influence, you can also declare the
//methods explicitly and provide additional code there with the standard initialization
//code. You can evaluate the return value.
METHOD FB_Init: BOOL
VAR_INPUT
    bInitRetains: BOOL; // TRUE: the retain variables are initialized (reset warm / reset cold)
    bInCopyCode: BOOL;  // TRUE: the instance will be copied to the copy code afterward (online change)
	
	i_ptrServices: POINTER TO ServiceContainer;
	i_ptrPanelMgr: POINTER TO PanelManager;	
END_VAR
VAR
	i: UINT;
	m_statesEnum: EProcessVariables;
END_VAR
m_ptrServices := i_ptrServices;
m_ptrPanelMgr := i_ptrPanelMgr;

// the panel manager serves as an observation of the buttons
m_ptrServices^.PtrStateTracker^.AddObservation(m_ptrPanelMgr);

// optionally, disable pre-/ postconditions
// m_ptrServices^.PtrProcessManager^.SetAllConditionsTrue();

// init process variable names
FOR i := ResiConst.ARR_MIN TO ResiConst.STATE_ARR_MAX DO
	m_statesEnum := i;
	i_ptrServices^.PtrStateTracker^.SetProcessVariableName(i, TO_STRING(m_statesEnum));
END_FOR
	
FC_InitAlarmTexts();
END_METHOD

ACTION ReadyLights:
m_ptrPanelMgr^.SetGreen(TRUE, T#500MS);
m_ptrPanelMgr^.SetRed(FALSE);
m_ptrPanelMgr^.SetWhite(FALSE);
END_ACTION

ACTION StoppingLights:
m_ptrPanelMgr^.SetGreen(FALSE);
m_ptrPanelMgr^.SetRed(TRUE, T#500MS);
m_ptrPanelMgr^.SetWhite(FALSE);
END_ACTION

TRANSITION TAbort:
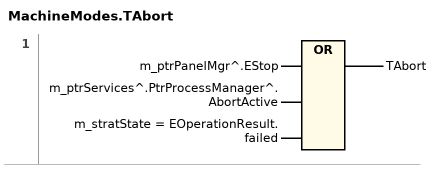
// NETWORK 1
TAbort := m_ptrPanelMgr^.EStop OR m_ptrServices^.PtrProcessManager^.AbortActive OR (m_stratState = EOperationResult.failed);
END_TRANSITION

END_FUNCTION_BLOCK
